Fanuc KAREL source: kx00011.KL

-- PROVISIONAL review KL for V940-1; original PC SHA256 56e006186fd9a42125a43de49b7953ac216d4a5ef88eada01bf3f257717129ab
-- Incomplete behavior may be omitted. Consult companion uncertainty JSON. Do not deploy.
PROGRAM KX00011
%NOLOCKGROUP
VAR
  I : INTEGER
  J : INTEGER
  B : BOOLEAN
  F : FILE
  S : STRING[80]
-- UNRESOLVED_DECL P type=000102
BEGIN
  -- V9_ZERO_TABLE_METADATA_HINT layout=0001; no indexed target words; source/name/runtime held
  -- UNRESOLVED_PC offsets 5-7; opcodes 9C,65
  -- UNRESOLVED_PC offsets 12-16; opcodes 7F
END KX00011
